TYPE CamOut_Param_typ :
	STRUCT
		Options 		: ST_GearOutOptions; //Currently not implemented/used
	END_STRUCT
END_TYPE

(* stored: Version 1.1.0.1, ProductVersion 3.1.4024.3
   DUT CamOut_Param_typ: Id {05b1b064-9c12-050f-2462-db785d50848f} *)
